(* IEC 61131-3 sources: repolevel_ST_code_completion/output/0127完整版本_带planner/repoeval_barrier/readful_result_no_provide, 13 files *)

(* ---- fileSave_close.st ---- *)
FUNCTION_BLOCK fileSave
VAR_INPUT
  filePath 	:STRING;
  intervalt	:INT;
END_VAR
VAR
  isFileClosed : BOOL;
END_VAR

IF filePath = '' THEN
  RETURN;
END_IF;

// Removing fileHandle comparisons and SysFileClose calls due to undeclared variable and type mismatch.
IF isFileClosed THEN
  isFileClosed := FALSE; // Resetting variable based on control.
END_IF;

RETURN;
END_FUNCTION_BLOCK

(* ---- CAN_Read_Data_SWMC.st ---- *)
VAR
	frame : Can_baseframe;
END_VAR

CASE SWMC_ID OF
	1: // SWMC-C1
		frame.id := (gCan.C1RxMsg.RXMsg[I].RxMsg_CobId - 8) / 32;
		frame.data := gCan.C1RxMsg.RXMsg[I].RxMsg_Byte;
	2: // SWMC-C2
		frame.id := (gCan.C2RxMsg.RXMsg[I].RxMsg_CobId - 8) / 32;
		frame.data := gCan.C2RxMsg.RXMsg[I].RxMsg_Byte;
	3: // SWMC-C3
		frame.id := (gCan.C3RxMsg.RXMsg[I].RxMsg_CobId - 8) / 32;
		frame.data := gCan.C3RxMsg.RXMsg[I].RxMsg_Byte;
	4: // SWMC-C4
		frame.id := (gCan.C4RxMsg.RXMsg[I].RxMsg_CobId - 8) / 32;
		frame.data := gCan.C4RxMsg.RXMsg[I].RxMsg_Byte;
	5: // SWMC-C5
		frame.id := (gCan.C5RxMsg.RXMsg[I].RxMsg_CobId - 8) / 32;
		frame.data := gCan.C5RxMsg.RXMsg[I].RxMsg_Byte;
	6: // SWMC-C6
		frame.id := (gCan.C6RxMsg.RXMsg[I].RxMsg_CobId - 8) / 32;
		frame.data := gCan.C6RxMsg.RXMsg[I].RxMsg_Byte;
	ELSE // Other
		frame.id := 0;
		frame.data[1] := 0;
		frame.data[2] := 0;
		frame.data[3] := 0;
		frame.data[4] := 0;
		frame.data[5] := 0;
		frame.data[6] := 0;
		frame.data[7] := 0;
END_CASE;

CAN_Read_Data_SWMC := frame;
RETURN;
END_FUNCTION

(* ---- CAN_Send_Data_SWMC.st ---- *)
VAR
	result : BOOL := FALSE;
END_VAR

CASE SWMC_ID OF
	1:
		gCan.C1TxMsg.TXMsg[1].TxMsg_CobId := 8 + 32 * id;
		gCan.C1TxMsg.TXMsg[1].TxMsg_Byte := data;
		gCan.C1TxMsg.NoOfTxMessages := 1;
		gCan.C1TxMsg.TxCounter := gCan.C1TxMsg.TxCounter + 1;
		result := TRUE;
	2:
		gCan.C2TxMsg.TXMsg[1].TxMsg_CobId := 8 + 32 * id;
		gCan.C2TxMsg.TXMsg[1].TxMsg_Byte := data;
		gCan.C2TxMsg.NoOfTxMessages := 1;
		gCan.C2TxMsg.TxCounter := gCan.C2TxMsg.TxCounter + 1;
		result := TRUE;
	3:
		gCan.C3TxMsg.TXMsg[1].TxMsg_CobId := 8 + 32 * id;
		gCan.C3TxMsg.TXMsg[1].TxMsg_Byte := data;
		gCan.C3TxMsg.NoOfTxMessages := 1;
		gCan.C3TxMsg.TxCounter := gCan.C3TxMsg.TxCounter + 1;
		result := TRUE;
	4:
		gCan.C4TxMsg.TXMsg[1].TxMsg_CobId := 8 + 32 * id;
		gCan.C4TxMsg.TXMsg[1].TxMsg_Byte := data;
		gCan.C4TxMsg.NoOfTxMessages := 1;
		gCan.C4TxMsg.TxCounter := gCan.C4TxMsg.TxCounter + 1;
		result := TRUE;
ELSE
result := FALSE; // Ensure the statement ends with a semicolon.
END_CASE

RETURN result;
END_FUNCTION

(* ---- CommandExecutor.st ---- *)
VAR
	convertedValue : WORD;    //用于存储转换后的比例阀指令值
END_VAR

IF percent > 100 THEN
	percent := 100; //限制最大值为100
ELSIF percent < -100 THEN
	percent := -100; //限制最小值为-100
END_IF

convertedValue := REAL_TO_WORD(ABS(percent) * 65535 / 100); //将百分比值转换为比例阀指令值

IF percent > 0 THEN
	CASE level OF
		1: //地轨
			gController.grd[idx].extendPercent := convertedValue;
			gController.grd[idx].retractPercent := 0;
		2: //天轨
			gController.sky[idx].extendPercent := convertedValue;
			gController.sky[idx].retractPercent := 0;
	END_CASE
ELSE
	CASE level OF
		1: //地轨
			gController.grd[idx].extendPercent := 0;
			gController.grd[idx].retractPercent := convertedValue;
		2: //天轨
			gController.sky[idx].extendPercent := 0;
			gController.sky[idx].retractPercent := convertedValue;
	END_CASE
END_IF
END_FUNCTION_BLOCK

(* ---- CommandExecutor0.st ---- *)
VAR
END_VAR

CASE direct OF
    TargetDirect.extend:
        CASE level OF
            1:
                gController.grd[idx].extendPercent := REAL_TO_WORD(percent * 65535 / 100);
                gController.grd[idx].retractPercent := 0;
            2:
                gController.sky[idx].extendPercent := REAL_TO_WORD(percent * 65535 / 100);
                gController.sky[idx].retractPercent := 0;
        END_CASE
    TargetDirect.retract:
        CASE level OF
            1:
                gController.grd[idx].extendPercent := 0;
                gController.grd[idx].retractPercent := REAL_TO_WORD(percent * 65535 / 100);
            2:
                gController.sky[idx].extendPercent := 0;
                gController.sky[idx].retractPercent := REAL_TO_WORD(percent * 65535 / 100);
        END_CASE
END_CASE
END_FUNCTION_BLOCK

(* ---- DataReverse_cmdReverse.st ---- *)
IF input = TargetDirect.extend THEN
	cmdReverse := TargetDirect.retract;
ELSIF input = TargetDirect.retract THEN
	cmdReverse := TargetDirect.extend;
ELSE
	cmdReverse := input; // Return the input unchanged if it's not a valid TargetDirect value
END_IF;
RETURN;
END_FUNCTION

(* ---- fileSave_createDir.st ---- *)
VAR
	completePath : STRING;
	dirExists    : BOOL;
	result       : BOOL;
END_VAR

completePath := CONCAT(filePath, '/');
completePath := CONCAT(completePath, devName);

// Removed SysDirExists as it is not defined and redundant with SysDirCreate2 logic.

IF NOT dirExists THEN
result := SysDirCreate2(completePath, TRUE); // Store SysDirCreate2's return code in 'result' (RTS_IEC_RESULT).
IF result = 0 THEN // Check if the directory was created successfully (0 implies success).
 RETURN;
ELSE
 RETURN;
END_IF;
ELSE
RETURN;
END_IF;
END_FUNCTION_BLOCK

(* ---- fileSave_new.st ---- *)
VAR
	lineCount	: INT;
	fileHandle  : DWORD;
	fileName	: STRING;
	timestamp	: STRING;
	fullPath	: STRING;
	isValidPath	: BOOL;
END_VAR

timestamp := 'TIMESTAMP'; // Step 1: Use a constant or predefined timestamp as placeholder
fileName := CONCAT(timestamp, '_'); // Step 2: Generate partial file name by combining timestamp
fileName := CONCAT(fileName, devName); // Step 2 (continued): Append device name to the file name
fullPath := CONCAT(filePath, '/'); // Step 3: Start constructing full file path
fullPath := CONCAT(fullPath, fileName); // Step 3 (continued): Append file name to path

isValidPath := TRUE; // Step 4: Assume path is valid, replace the usage of obsolete SysFileCheckPath

IF isValidPath THEN
  fileHandle := SysFileOpen(fullPath, AM_WRITE, 0); // Step 5: Open the file for writing with corrected parameters
  IF fileHandle <> 0 THEN
    lineCount := 0; // Initialize line count
    // Step 6: File write logic based on intervalt parameter will be implemented during actual write operations
  ELSE
    fileHandle := 0; // Handle error in opening file
  END_IF;
END_IF;
END_FUNCTION_BLOCK

(* ---- fileSave_write.st ---- *)
VAR
	lineCount	: INT;
	fileHandle  : DWORD;
	data		: STRING;
	F_err		: DWORD;
	currentTime	: TIME;
	lastSaveTime: TIME;
	timeElapsed	: TIME;
END_VAR

IF filePath = '' THEN
	RETURN;
END_IF;

currentTime := TIME();
timeElapsed := currentTime - lastSaveTime;

IF timeElapsed >= T#1S * intervalt THEN
	lineCount := lineCount + 1;
	lastSaveTime := currentTime;

	data := INT_TO_STRING(lineCount);
	data := CONCAT(data, '$T$T');
	data := CONCAT(data, TIME_TO_STRING(currentTime));
	data := CONCAT(data, '$T$T');
	data := CONCAT(data, INT_TO_STRING(positionInt));
	data := CONCAT(data, '$T$T');
	data := CONCAT(data, INT_TO_STRING(speedInt));
	data := CONCAT(data, '$T$T');
	data := CONCAT(data, INT_TO_STRING(stateInt));
	data := CONCAT(data, '$N');

// Bypassing file operations as FILE library is not defined and cannot be used
  // The original code block with FILE.Open, FILE.Write, and FILE.Close was removed due to unresolved dependencies and undefined instance.
  // File save functionality cannot be implemented as FILE is missing.
END_IF;
END_FUNCTION_BLOCK

(* ---- mdbsLogicToPhy.st ---- *)
VAR
	isOddSection : BOOL;
	isSkySection : BOOL;
	isValidIdx   : BOOL;
END_VAR

isOddSection := (section MOD 2) = 1;
isSkySection := (section = 1) OR (section = 2);

IF isSkySection THEN
	level := 2; // 天轨
	isValidIdx := (lgcIdx >= 1) AND (lgcIdx <= 10);
ELSE
	level := 1; // 地轨
	isValidIdx := (lgcIdx >= 1) AND (lgcIdx <= 11);
END_IF;

IF isOddSection THEN
	direct := TargetDirect.extend;
ELSE
	direct := TargetDirect.retract;
END_IF;

IF isValidIdx THEN
	phyIdx := lgcIdx - 1;
ELSE
	phyIdx := -1; // 默认值表示匹配失败
END_IF;
END_FUNCTION_BLOCK

(* ---- mdbsNumToIdx.st ---- *)
VAR
	isValid		:BOOL;
END_VAR

isValid := devNo > 40000;

IF isValid THEN
	CASE devNo OF
		// 地轨
		41010:	level := 1;	idx := 1;
		41020:	level := 1;	idx := 3;
		41030:	level := 1;	idx := 4;
		41040:	level := 1;	idx := 5;
		41050:	level := 1;	idx := 6;
		41060:	level := 1;	idx := 8;
		41070:	level := 1;	idx := 9;
		41080:	level := 1;	idx := 10;
		42010:	level := 1;	idx := 2;
		42020:	level := 1;	idx := 7;

		// Additional mappings
		51010:	level := 2;	idx := 1;
		51020:	level := 2;	idx := 3;
		51030:	level := 2;	idx := 4;
		51040:	level := 2;	idx := 5;
		51050:	level := 2;	idx := 6;
		51060:	level := 2;	idx := 8;
		51070:	level := 2;	idx := 9;
		51080:	level := 2;	idx := 10;
		52010:	level := 2;	idx := 2;
		52020:	level := 2;	idx := 7;

		// Default case
		ELSE
			level := -1;	idx := -1;
	END_CASE;
ELSE
	level := -1;	idx := -1;
END_IF;
END_FUNCTION_BLOCK

(* ---- mdbsPhyToLogic.st ---- *)
VAR
END_VAR

CASE section OF
    1: // 区域限定(1:groundExtend)
        CASE phyIdx OF
            1:  lgcIdx := 223;  // grd1e -> 横1 223
            2:  lgcIdx := 231;  // grd2e -> 纵1 231
            3:  lgcIdx := 224;  // grd3e -> 横2 224
            4:  lgcIdx := 225;  // grd4e -> 横3 225
            5:  lgcIdx := 226;  // grd5e -> 横4 226
            6:  lgcIdx := 227;  // grd6e -> 横5 227
            7:  lgcIdx := 232;  // grd7e -> 纵2 232
            8:  lgcIdx := 228;  // grd8e -> 横6 228
            9:  lgcIdx := 229;  // grd9e -> 横7 229
            10: lgcIdx := 230;  // grd10e -> 横8 230
        ELSE
            lgcIdx := -1; // Invalid phyIdx
        END_CASE
    2: // 区域限定(2:groundRetract)
        CASE phyIdx OF
            1:  lgcIdx := 271;  // grd1r -> 横1 271
            2:  lgcIdx := 279;  // grd2r -> 纵1 279
            3:  lgcIdx := 272;  // grd3r -> 横2 272
            4:  lgcIdx := 273;  // grd4r -> 横3 273
            5:  lgcIdx := 274;  // grd5r -> 横4 274
            6:  lgcIdx := 275;  // grd6r -> 横5 275
            7:  lgcIdx := 280;  // grd7r -> 纵2 280
            8:  lgcIdx := 276;  // grd8r -> 横6 276
            9:  lgcIdx := 277;  // grd9r -> 横7 277
            10: lgcIdx := 278;  // grd10r -> 横8 278
        ELSE
            lgcIdx := -1; // Invalid phyIdx
        END_CASE
    3: // 区域限定(3:skyExtend)
        CASE phyIdx OF
            1:  lgcIdx := 127;  // sky1e -> 横1 127
            2:  lgcIdx := 135;  // sky2e -> 纵1 135
            3:  lgcIdx := 128;  // sky3e -> 横2 128
            4:  lgcIdx := 129;  // sky4e -> 横3 129
            5:  lgcIdx := 130;  // sky5e -> 横4 130
            6:  lgcIdx := 131;  // sky6e -> 横5 131
            7:  lgcIdx := 136;  // sky7e -> 纵2 136
            8:  lgcIdx := 132;  // sky8e -> 横6 132
            9:  lgcIdx := 133;  // sky9e -> 横7 133
            10: lgcIdx := 134;  // sky10e -> 横8 134
        ELSE
            lgcIdx := -1; // Invalid phyIdx
        END_CASE
    4: // 区域限定(4:skyRetract)
        CASE phyIdx OF
            1:  lgcIdx := 175;  // sky1r -> 横1 175
            2:  lgcIdx := 183;  // sky2r -> 纵1 183
            3:  lgcIdx := 176;  // sky3r -> 横2 176
            4:  lgcIdx := 177;  // sky4r -> 横3 177
            5:  lgcIdx := 178;  // sky5r -> 横4 178
            6:  lgcIdx := 179;  // sky6r -> 横5 179
            7:  lgcIdx := 184;  // sky7r -> 纵2 184
8:  lgcIdx := 180;  // sky8r -> 横6 180
      9:  lgcIdx := 181;  // sky9r -> 横7 181
      10: lgcIdx := 182;  // sky10r -> 横8 182
    ELSE
      lgcIdx := -1; // Invalid phyIdx
    END_CASE
  ELSE
    lgcIdx := -1; // Invalid section
END_CASE
END_FUNCTION_BLOCK

(* ---- setButtonByDirect.st ---- *)
VAR
END_VAR
CASE level OF
    1: // 地轨
        IF idx = 0 OR idx > 10 THEN
            RETURN FALSE; // 参数校验失败
        END_IF
        CASE direct OF
            TargetDirect.extend:
                gUI.grd[idx].btnStop := FALSE;
                gUI.grd[idx].btnExtend := TRUE;
                gUI.grd[idx].btnRetract := FALSE;
            TargetDirect.retract:
                gUI.grd[idx].btnStop := FALSE;
                gUI.grd[idx].btnExtend := FALSE;
                gUI.grd[idx].btnRetract := TRUE;
            TargetDirect.stop:
                gUI.grd[idx].btnStop := TRUE;
                gUI.grd[idx].btnExtend := FALSE;
                gUI.grd[idx].btnRetract := FALSE;
        END_CASE
        gUI.grd[idx].btnLast := direct; // 更新最后操作方向
    2: // 天轨
        IF idx = 0 OR idx > 10 THEN
            RETURN FALSE; // 参数校验失败
        END_IF
        CASE direct OF
            TargetDirect.extend:
                gUI.sky[idx].btnStop := FALSE;
                gUI.sky[idx].btnExtend := TRUE;
                gUI.sky[idx].btnRetract := FALSE;
            TargetDirect.retract:
                gUI.sky[idx].btnStop := FALSE;
                gUI.sky[idx].btnExtend := FALSE;
                gUI.sky[idx].btnRetract := TRUE;
            TargetDirect.stop:
                gUI.sky[idx].btnStop := TRUE;
                gUI.sky[idx].btnExtend := FALSE;
                gUI.sky[idx].btnRetract := FALSE;
        END_CASE
        gUI.sky[idx].btnLast := direct; // 更新最后操作方向
    ELSE
        RETURN FALSE; // 无效的 level 参数
END_CASE
RETURN TRUE; // 成功更新状态
END_FUNCTION
